PROGRAM MAIN
VAR
END_VAR

Control_SFC();

END_PROGRAM

(* stored: Version 1.1.0.1, ProductVersion 3.1.4024.12
   POU MAIN: Id {c6f84632-701f-4f7b-9b68-bc8966d9fa81}, SpecialFunc None *)
